FUNCTION_BLOCK FieldsToArrowheadCloud (* Translate individual fields to an ArrowheadCloud type *)
  (* Standard: 61499-2; Description: Copyright (c) 2018 fortiss GmbH This program and the accompanying materials are made available under the terms of the Eclipse Public License 2.0 which is available at https://www.eclipse.org/legal/epl-2.0/ SPDX-License-Identifier: EPL-2.0 *)
  (* Version 1.0, 2018-09-21, Jose Cabral, fortiss GmbH *)
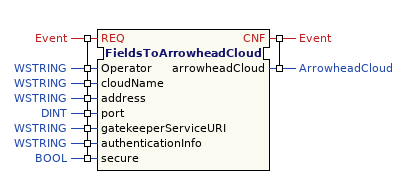
  EVENT_INPUT
    REQ WITH Operator, cloudName, address, secure, authenticationInfo, gatekeeperServiceURI, port; (* Create arrowhead cloud *)
  END_EVENT
  EVENT_OUTPUT
    CNF WITH arrowheadCloud; (* Arrowhead cloud created *)
  END_EVENT
  VAR_INPUT
    Operator : WSTRING; (* Company (the capital  O is to avoid clash when exporting to C++) *)
    cloudName : WSTRING; (* Identification of the cloud *)
    address : WSTRING; (* Address to access the cloud *)
    port : DINT; (* Port to access the cloud *)
    gatekeeperServiceURI : WSTRING; (* (Unclear documentation) *)
    authenticationInfo : WSTRING; (* Authentication info of the cloud *)
    secure : BOOL; (* (Unclear documentation) *)
  END_VAR
  VAR_OUTPUT
    arrowheadCloud : ArrowheadCloud; (* Created Arrowhead cloud *)
  END_VAR
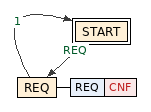
  EC_STATES
    START; (* Initial State *)
    REQ : REQ -> CNF; (* Normal execution *)
  END_STATES
  EC_TRANSITIONS
    START TO REQ := REQ;
    REQ TO START := 1;
  END_TRANSITIONS
  ALGORITHM REQ IN ST: (* Normally executed algorithm *)
arrowheadCloud.Operator := Operator;
arrowheadCloud.cloudName := cloudName;
arrowheadCloud.address := address;
arrowheadCloud.port := port;
arrowheadCloud.gatekeeperServiceURI := gatekeeperServiceURI;
arrowheadCloud.authenticationInfo := authenticationInfo;
arrowheadCloud.secure := secure;
  END_ALGORITHM
END_FUNCTION_BLOCK
